INTERFACE I_SingleDirectionMotor

METHOD PUBLIC Start
VAR_INPUT
END_VAR
END_METHOD

METHOD PUBLIC Stop
VAR_INPUT
END_VAR
END_METHOD

END_INTERFACE

(* stored: Version 1.1.0.1, ProductVersion 3.1.4024.11
   Itf I_SingleDirectionMotor: Id {6a980a69-0144-44cb-9910-de4cb72bdee3}
   Method Start: Id {a16f548e-bb80-4fc9-a8b5-6745645587aa}
   Method Stop: Id {3b779767-5501-4c72-b881-dd6db9c31389} *)
